ABB RobotStudio station: EstacionTaladrado.rsstn

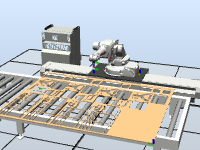
Station TEST_OPC (saved by RobotStudio 6.8.8307.1040)
Controller IRB1600APM, task T_ROB1: task frame (RAPID world) sits at (108, -475.5, 460) mm, rotated rx 0 ry 0 rz 90 deg in the station
Controller IRB1600APM
  mechanical unit ROB_1: IRB1600_6_145__02_5, 6 joints, base frame (0, 0, 0) mm
  mechanical unit TRACK_1: IRBT2005_IRB_STD_INT_0_0_3__01, 1 joints, base frame (0, 0, 0) mm
Layout (positions relative to the parent item):
  - Ventosa [mechanism, from Libraries\Ventosa.rslib] at (-1299.78, -50.5, 1120.91) mm, rotated rx -180 ry 0 rz 0 deg
  - Placa_de_Corte [part] at (-2250, -1220, 450) mm
  - IRC5_Singel-Cabinet [part, from Equipment\IRC5_Singel-Cabinet.rslib] at (1200, 1600, 100) mm, rotated rx 90 ry 0 rz 90 deg
  - 1320_4000_h2 [part, from Equipment\Conveyor 1320 4000 h2.rslib] at (-1985, 2600, 0) mm, rotated rx 0 ry 0 rz -90 deg
  - PLACA_SOPORTE_1 [part] at (-1199.98, 989.79, 462) mm, rotated rx -180 ry 0 rz -2.32 deg
  - IRB1600_6_145__02_5 [mechanism, from Robots\IRB1600_6_145_G_02.rslib] at (108, -50.5, 460) mm, rotated rx 0 ry 0 rz 90 deg; joint values [1.5708, 1.2217, -1.2217, 0, 1.5708, 0] (rad or m)
  - IRBT2005_IRB_STD_INT_0_0_3__01 [mechanism] at (400, -1300, 0) mm, rotated rx 0 ry 0 rz 90 deg; joint values [0.425] (rad or m)
      links: Base, Link1
  - Attacher [smart component, from Components\Attacher.rslib]
      properties: Parent=Ventosa; Flange=0; Child=PLACA_SOPORTE_1; Mount=true; Offset=[0 0 0]; Orientation=[0 0 0]
  - Detacher [smart component, from Components\Detacher.rslib]
      properties: Child=PLACA_SOPORTE_1; KeepPosition=true
  - LogicGate_4 [smart component, from Components\LogicGate.rslib]
      properties: Operator=NOT; Delay=0
Attachment: IRB1600_6_145__02_5 is attached to IRBT2005_IRB_STD_INT_0_0_3__01 / Link1
Attachment: Ventosa is attached to IRB1600_6_145__02_5 / Link6
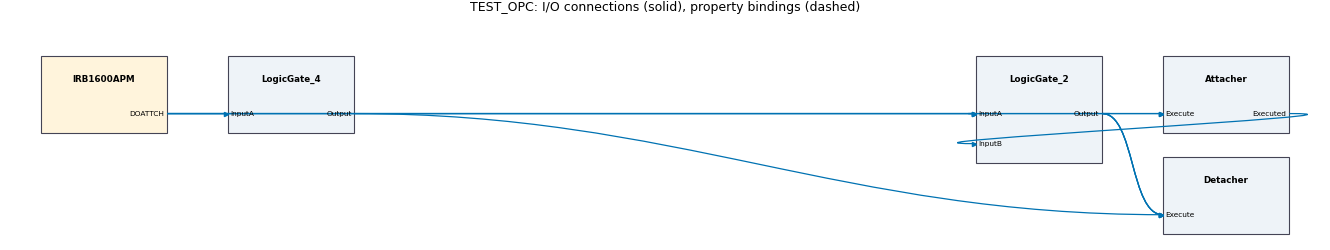
Station logic (signal -> signal, property => property):
  IRB1600APM.DOATTCH -> LogicGate_2.InputA
  LogicGate_2.Output -> LogicGate.InputA
  Attacher.Executed -> LogicGate.InputB
  LogicGate.Output -> Detacher.Execute
  LogicGate_2.Output -> Detacher.Execute
  LogicGate_3.Output -> Detacher.Execute
  LogicGate_3.Output -> Attacher.Execute
  IRB1600APM.DOATTCH -> LogicGate_3.InputA
  IRB1600APM.DOATTCH -> LogicGate_4.InputA
  LogicGate_4.Output -> Detacher.Execute
  IRB1600APM.DOATTCH -> Attacher.Execute
Targets, tools, work objects and paths stored in the station, written as RAPID:
! task T_ROB1
MODULE CalibData
  PERS tooldata VentosaTCP:=[TRUE,[[0,0,110.772],[1,0,0,0]],[1,[0,0,53.582],[1,0,0,0],0,0,0]];
  TASK PERS wobjdata Placa:=[FALSE,TRUE,"",[[0,0,0],[1,0,0,0]],[[-744.5,2358,-10],[0.707106781,0,0,-0.707106781]]];
ENDMODULE

! task T_ROB1
MODULE Module1
  CONST jointtarget MID_POINT:=[[90,70,-70,0,90,0],[425,9E+09,9E+09,9E+09,9E+09,9E+09]];
  CONST robtarget PLACA_SOPORTE_1:=[[1050.01804282,2209.787180675,12.000031193],[-0.000000003,0.999795002,-0.020247298,0.000000052],[0,-1,-1,0],[1350,9E+09,9E+09,9E+09,9E+09,9E+09]];
  PROC Path_MID_POINT()
    MoveAbsJ MID_POINT,v1000,z100,VentosaTCP\WObj:=Placa;
  ENDPROC
  PROC Path_PLACA_SOPORTE_1()
    MoveJ PLACA_SOPORTE_1,v1000,z100,VentosaTCP\WObj:=Placa;
  ENDPROC
ENDMODULE

